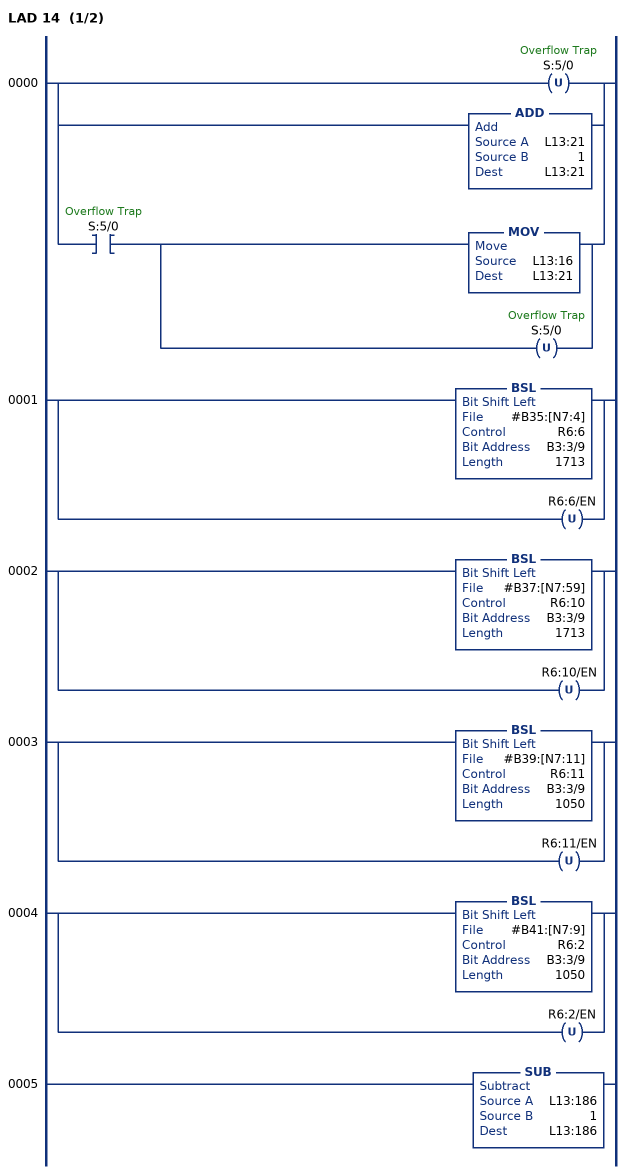
% Rung: 0 %
SOR BST OTU S:5/0 NXB ADD L13:21 1 L13:21 NXB XIC S:5/0 BST MOV L13:16 L13:21 NXB OTU S:5/0 BND BND EOR
%   S:5/0  "Overflow Trap" %
% Rung: 1 %
SOR BST BSL #B35:[N7:4] R6:6 B3:3/9 1713 NXB OTU R6:6/EN BND EOR
% Rung: 2 %
SOR BST BSL #B37:[N7:59] R6:10 B3:3/9 1713 NXB OTU R6:10/EN BND EOR
% Rung: 3 %
SOR BST BSL #B39:[N7:11] R6:11 B3:3/9 1050 NXB OTU R6:11/EN BND EOR
% Rung: 4 %
SOR BST BSL #B41:[N7:9] R6:2 B3:3/9 1050 NXB OTU R6:2/EN BND EOR
% Rung: 5 %
SOR SUB L13:186 1 L13:186 EOR

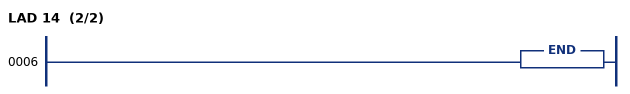
% Rung: 6 %
SOR END EOR

LADDER 81
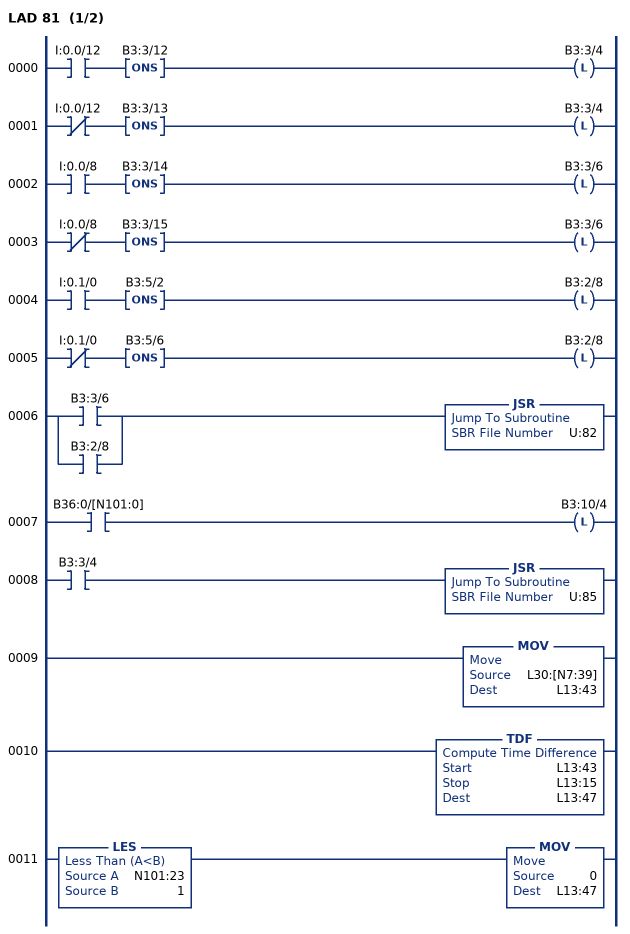
% Rung: 0 %
SOR XIC I:0.0/12 ONS B3:3/12 OTL B3:3/4 EOR
% Rung: 1 %
SOR XIO I:0.0/12 ONS B3:3/13 OTL B3:3/4 EOR
% Rung: 2 %
SOR XIC I:0.0/8 ONS B3:3/14 OTL B3:3/6 EOR
% Rung: 3 %
SOR XIO I:0.0/8 ONS B3:3/15 OTL B3:3/6 EOR
% Rung: 4 %
SOR XIC I:0.1/0 ONS B3:5/2 OTL B3:2/8 EOR
% Rung: 5 %
SOR XIO I:0.1/0 ONS B3:5/6 OTL B3:2/8 EOR
% Rung: 6 %
SOR BST XIC B3:3/6 NXB XIC B3:2/8 BND JSR U:82 EOR
% Rung: 7 %
SOR XIC B36:0/[N101:0] OTL B3:10/4 EOR
% Rung: 8 %
SOR XIC B3:3/4 JSR U:85 EOR
% Rung: 9 %
SOR MOV L30:[N7:39] L13:43 EOR
% Rung: 10 %
SOR TDF L13:43 L13:15 L13:47 EOR
% Rung: 11 %
SOR LES N101:23 1 MOV 0 L13:47 EOR

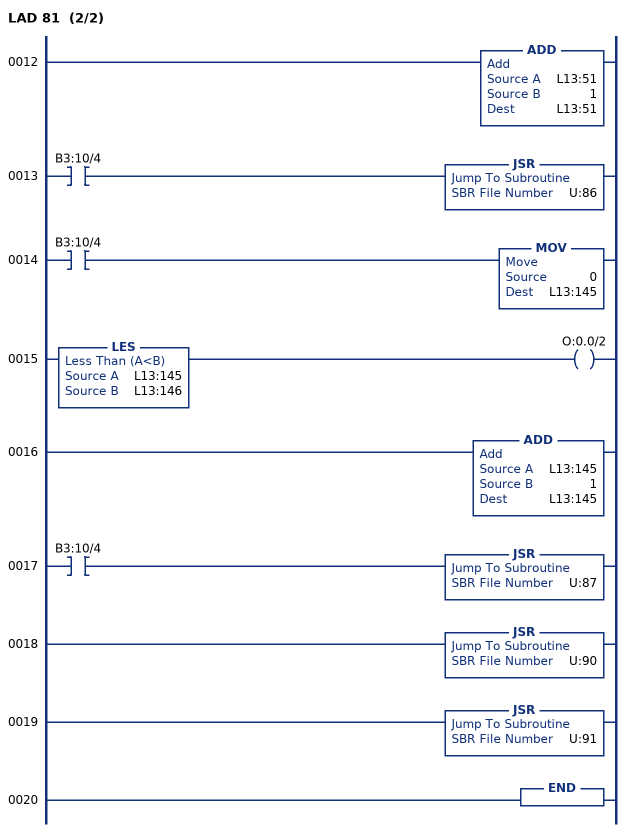
% Rung: 12 %
SOR ADD L13:51 1 L13:51 EOR
% Rung: 13 %
SOR XIC B3:10/4 JSR U:86 EOR
% Rung: 14 %
SOR XIC B3:10/4 MOV 0 L13:145 EOR
% Rung: 15 %
SOR LES L13:145 L13:146 OTE O:0.0/2 EOR
% Rung: 16 %
SOR ADD L13:145 1 L13:145 EOR
% Rung: 17 %
SOR XIC B3:10/4 JSR U:87 EOR
% Rung: 18 %
SOR JSR U:90 EOR
% Rung: 19 %
SOR JSR U:91 EOR
% Rung: 20 %
SOR END EOR

LADDER 82
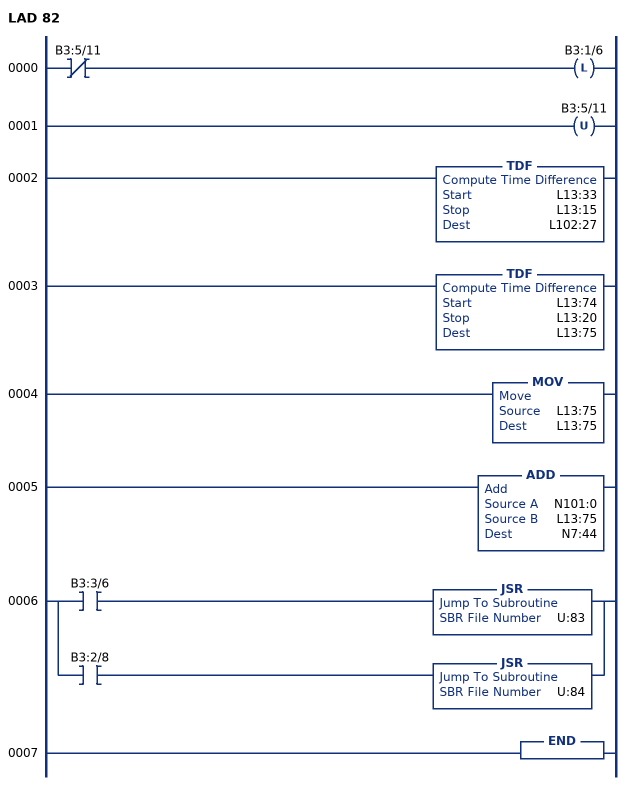
% Rung: 0 %
SOR XIO B3:5/11 OTL B3:1/6 EOR
% Rung: 1 %
SOR OTU B3:5/11 EOR
% Rung: 2 %
SOR TDF L13:33 L13:15 L102:27 EOR
% Rung: 3 %
SOR TDF L13:74 L13:20 L13:75 EOR
% Rung: 4 %
SOR MOV L13:75 L13:75 EOR
% Rung: 5 %
SOR ADD N101:0 L13:75 N7:44 EOR
% Rung: 6 %
SOR BST XIC B3:3/6 JSR U:83 NXB XIC B3:2/8 JSR U:84 BND EOR
% Rung: 7 %
SOR END EOR

LADDER 83
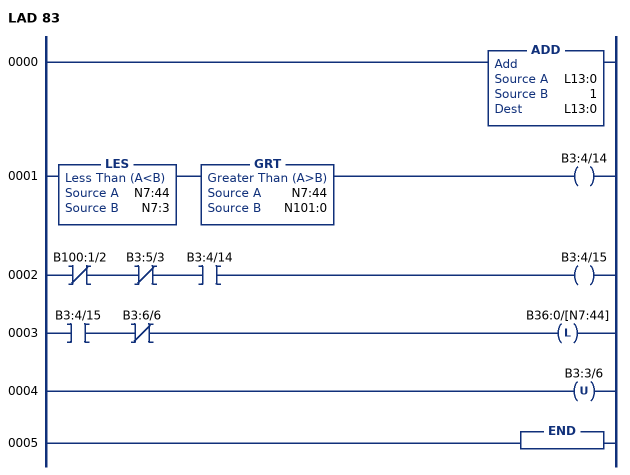
% Rung: 0 %
SOR ADD L13:0 1 L13:0 EOR
% Rung: 1 %
SOR LES N7:44 N7:3 GRT N7:44 N101:0 OTE B3:4/14 EOR
% Rung: 2 %
SOR XIO B100:1/2 XIO B3:5/3 XIC B3:4/14 OTE B3:4/15 EOR
% Rung: 3 %
SOR XIC B3:4/15 XIO B3:6/6 OTL B36:0/[N7:44] EOR
% Rung: 4 %
SOR OTU B3:3/6 EOR
% Rung: 5 %
SOR END EOR

LADDER 84
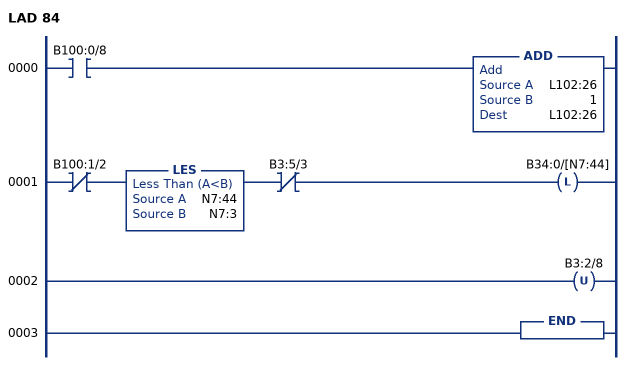
% Rung: 0 %
SOR XIC B100:0/8 ADD L102:26 1 L102:26 EOR
% Rung: 1 %
SOR XIO B100:1/2 LES N7:44 N7:3 XIO B3:5/3 OTL B34:0/[N7:44] EOR
% Rung: 2 %
SOR OTU B3:2/8 EOR
% Rung: 3 %
SOR END EOR

LADDER 85
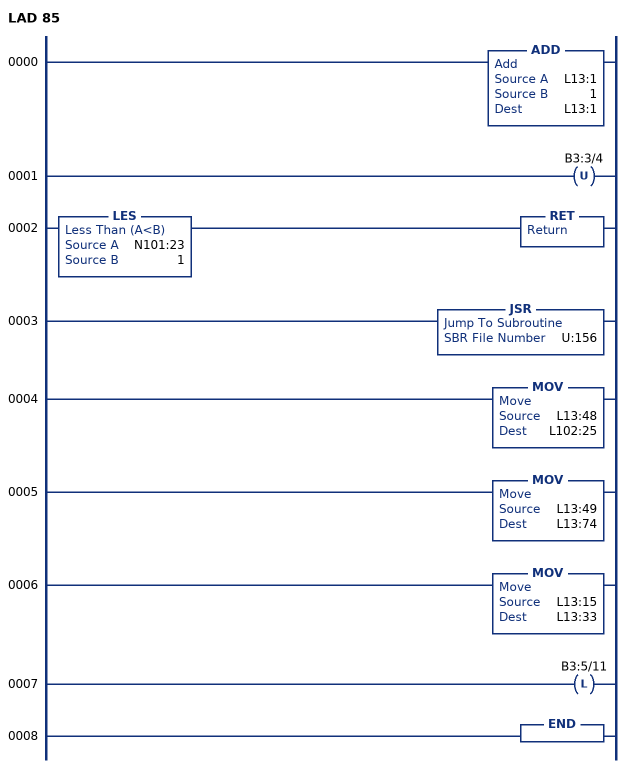
% Rung: 0 %
SOR ADD L13:1 1 L13:1 EOR
% Rung: 1 %
SOR OTU B3:3/4 EOR
% Rung: 2 %
SOR LES N101:23 1 RET EOR
% Rung: 3 %
SOR JSR U:156 EOR
% Rung: 4 %
SOR MOV L13:48 L102:25 EOR
% Rung: 5 %
SOR MOV L13:49 L13:74 EOR
% Rung: 6 %
SOR MOV L13:15 L13:33 EOR
% Rung: 7 %
SOR OTL B3:5/11 EOR
% Rung: 8 %
SOR END EOR

LADDER 86
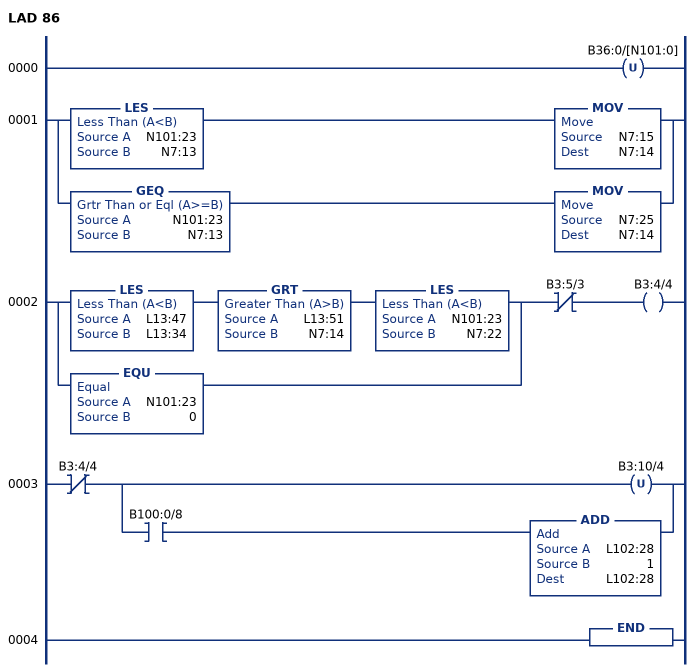
% Rung: 0 %
SOR OTU B36:0/[N101:0] EOR
% Rung: 1 %
SOR BST LES N101:23 N7:13 MOV N7:15 N7:14 NXB GEQ N101:23 N7:13 MOV N7:25 N7:14 BND EOR
% Rung: 2 %
SOR BST LES L13:47 L13:34 GRT L13:51 N7:14 LES N101:23 N7:22 NXB EQU N101:23 0 BND XIO B3:5/3 OTE B3:4/4 EOR
% Rung: 3 %
SOR XIO B3:4/4 BST OTU B3:10/4 NXB XIC B100:0/8 ADD L102:28 1 L102:28 BND EOR
% Rung: 4 %
SOR END EOR

LADDER 87
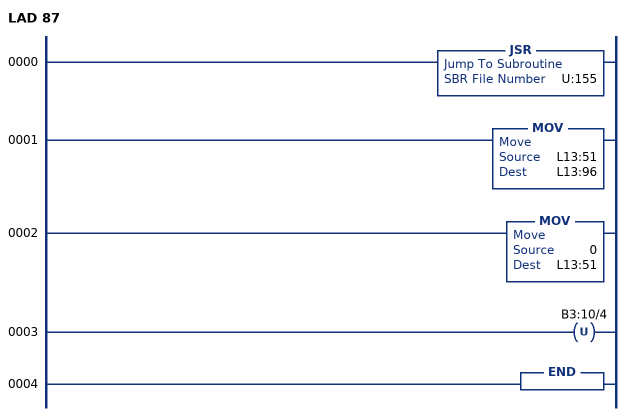
% Rung: 0 %
SOR JSR U:155 EOR
% Rung: 1 %
SOR MOV L13:51 L13:96 EOR
% Rung: 2 %
SOR MOV 0 L13:51 EOR
% Rung: 3 %
SOR OTU B3:10/4 EOR
% Rung: 4 %
SOR END EOR

LADDER 90
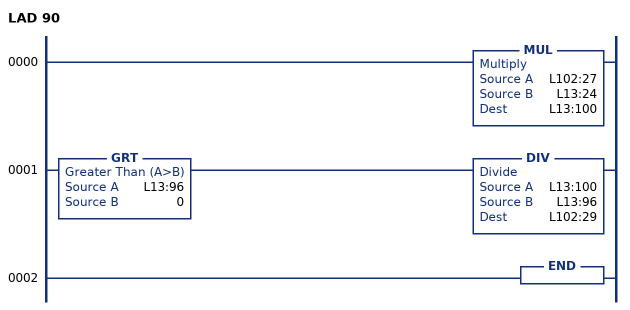
% Rung: 0 %
SOR MUL L102:27 L13:24 L13:100 EOR
% Rung: 1 %
SOR GRT L13:96 0 DIV L13:100 L13:96 L102:29 EOR
% Rung: 2 %
SOR END EOR

LADDER 91
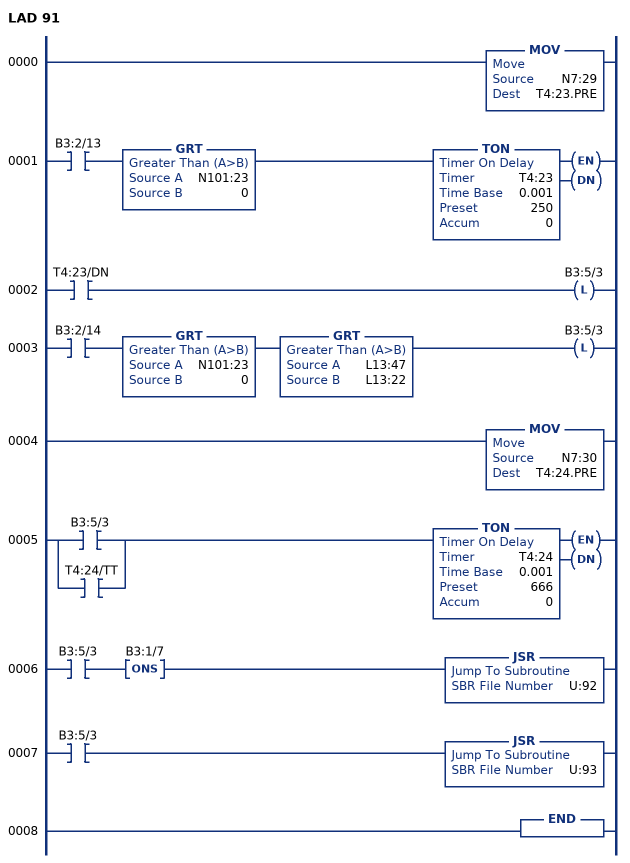
% Rung: 0 %
SOR MOV N7:29 T4:23.PRE EOR
% Rung: 1 %
SOR XIC B3:2/13 GRT N101:23 0 TON T4:23 0.001 250 0 EOR
% Rung: 2 %
SOR XIC T4:23/DN OTL B3:5/3 EOR
% Rung: 3 %
SOR XIC B3:2/14 GRT N101:23 0 GRT L13:47 L13:22 OTL B3:5/3 EOR
% Rung: 4 %
SOR MOV N7:30 T4:24.PRE EOR
% Rung: 5 %
SOR BST XIC B3:5/3 NXB XIC T4:24/TT BND TON T4:24 0.001 666 0 EOR
% Rung: 6 %
SOR XIC B3:5/3 ONS B3:1/7 JSR U:92 EOR
% Rung: 7 %
SOR XIC B3:5/3 JSR U:93 EOR
% Rung: 8 %
SOR END EOR

LADDER 92
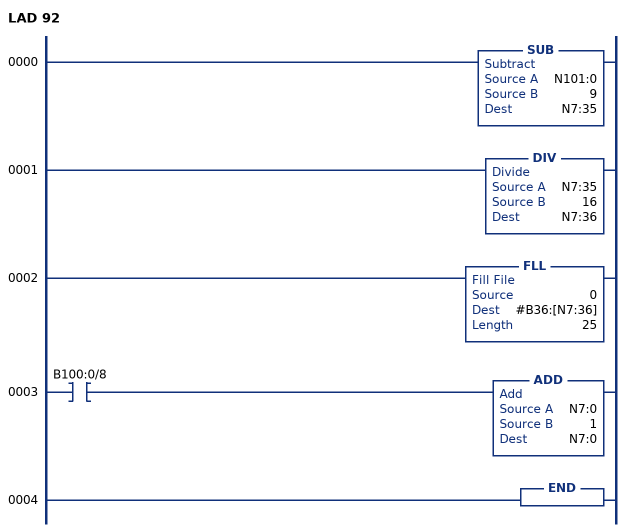
% Rung: 0 %
SOR SUB N101:0 9 N7:35 EOR
% Rung: 1 %
SOR DIV N7:35 16 N7:36 EOR
% Rung: 2 %
SOR FLL 0 #B36:[N7:36] 25 EOR
% Rung: 3 %
SOR XIC B100:0/8 ADD N7:0 1 N7:0 EOR
% Rung: 4 %
SOR END EOR

LADDER 93
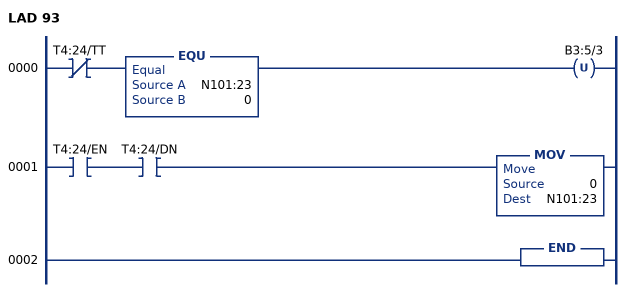
% Rung: 0 %
SOR XIO T4:24/TT EQU N101:23 0 OTU B3:5/3 EOR
% Rung: 1 %
SOR XIC T4:24/EN XIC T4:24/DN MOV 0 N101:23 EOR
% Rung: 2 %
SOR END EOR

LADDER 94
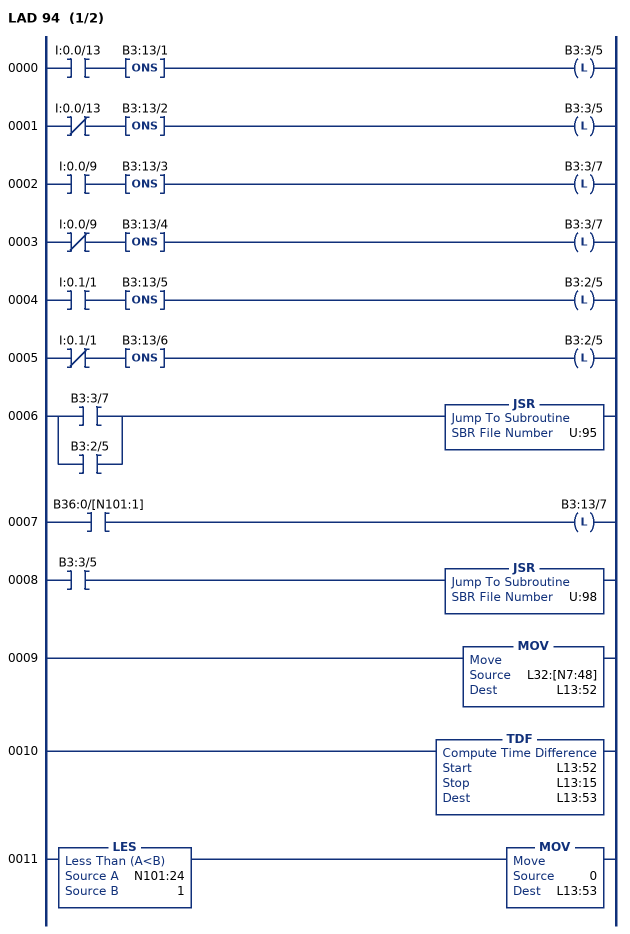
% Rung: 0 %
SOR XIC I:0.0/13 ONS B3:13/1 OTL B3:3/5 EOR
% Rung: 1 %
SOR XIO I:0.0/13 ONS B3:13/2 OTL B3:3/5 EOR
% Rung: 2 %
SOR XIC I:0.0/9 ONS B3:13/3 OTL B3:3/7 EOR
% Rung: 3 %
SOR XIO I:0.0/9 ONS B3:13/4 OTL B3:3/7 EOR
% Rung: 4 %
SOR XIC I:0.1/1 ONS B3:13/5 OTL B3:2/5 EOR
% Rung: 5 %
SOR XIO I:0.1/1 ONS B3:13/6 OTL B3:2/5 EOR
% Rung: 6 %
SOR BST XIC B3:3/7 NXB XIC B3:2/5 BND JSR U:95 EOR
% Rung: 7 %
SOR XIC B36:0/[N101:1] OTL B3:13/7 EOR
% Rung: 8 %
SOR XIC B3:3/5 JSR U:98 EOR
% Rung: 9 %
SOR MOV L32:[N7:48] L13:52 EOR
% Rung: 10 %
SOR TDF L13:52 L13:15 L13:53 EOR
% Rung: 11 %
SOR LES N101:24 1 MOV 0 L13:53 EOR

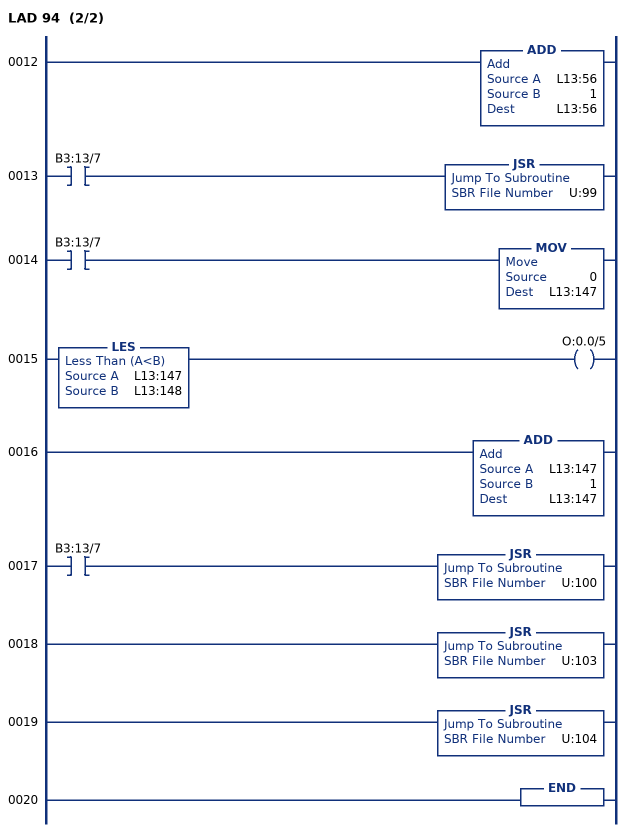
% Rung: 12 %
SOR ADD L13:56 1 L13:56 EOR
% Rung: 13 %
SOR XIC B3:13/7 JSR U:99 EOR
% Rung: 14 %
SOR XIC B3:13/7 MOV 0 L13:147 EOR
% Rung: 15 %
SOR LES L13:147 L13:148 OTE O:0.0/5 EOR
% Rung: 16 %
SOR ADD L13:147 1 L13:147 EOR
% Rung: 17 %
SOR XIC B3:13/7 JSR U:100 EOR
% Rung: 18 %
SOR JSR U:103 EOR
% Rung: 19 %
SOR JSR U:104 EOR
% Rung: 20 %
SOR END EOR

LADDER 95
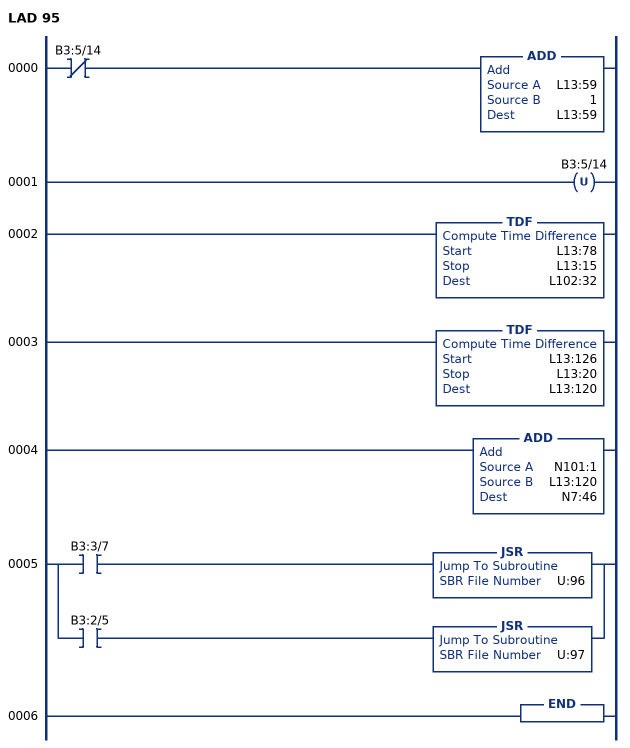
% Rung: 0 %
SOR XIO B3:5/14 ADD L13:59 1 L13:59 EOR
% Rung: 1 %
SOR OTU B3:5/14 EOR
% Rung: 2 %
SOR TDF L13:78 L13:15 L102:32 EOR
% Rung: 3 %
SOR TDF L13:126 L13:20 L13:120 EOR
% Rung: 4 %
SOR ADD N101:1 L13:120 N7:46 EOR
% Rung: 5 %
SOR BST XIC B3:3/7 JSR U:96 NXB XIC B3:2/5 JSR U:97 BND EOR
% Rung: 6 %
SOR END EOR

LADDER 96
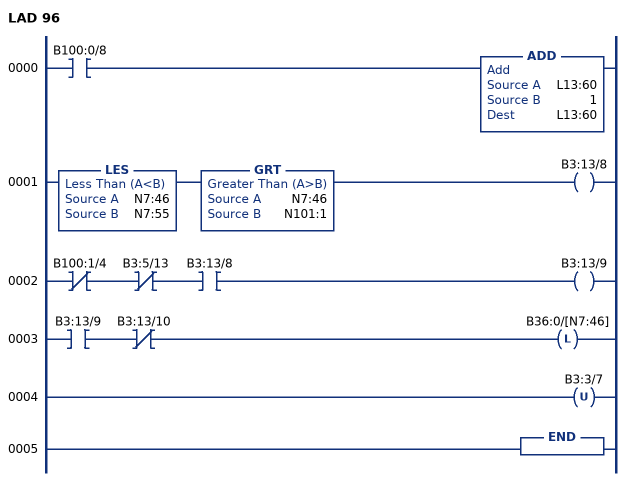
% Rung: 0 %
SOR XIC B100:0/8 ADD L13:60 1 L13:60 EOR
% Rung: 1 %
SOR LES N7:46 N7:55 GRT N7:46 N101:1 OTE B3:13/8 EOR
% Rung: 2 %
SOR XIO B100:1/4 XIO B3:5/13 XIC B3:13/8 OTE B3:13/9 EOR
% Rung: 3 %
SOR XIC B3:13/9 XIO B3:13/10 OTL B36:0/[N7:46] EOR
% Rung: 4 %
SOR OTU B3:3/7 EOR
% Rung: 5 %
SOR END EOR

LADDER 97
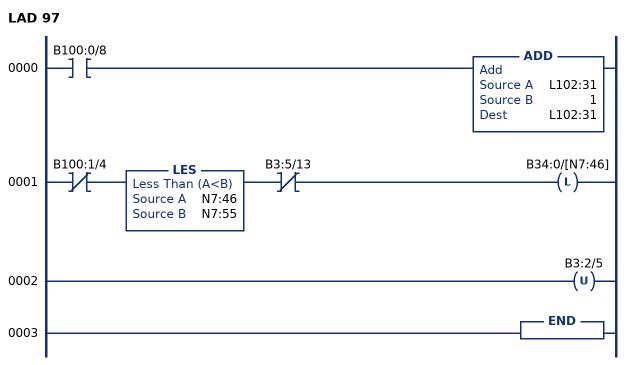
% Rung: 0 %
SOR XIC B100:0/8 ADD L102:31 1 L102:31 EOR
% Rung: 1 %
SOR XIO B100:1/4 LES N7:46 N7:55 XIO B3:5/13 OTL B34:0/[N7:46] EOR
% Rung: 2 %
SOR OTU B3:2/5 EOR
% Rung: 3 %
SOR END EOR

LADDER 98
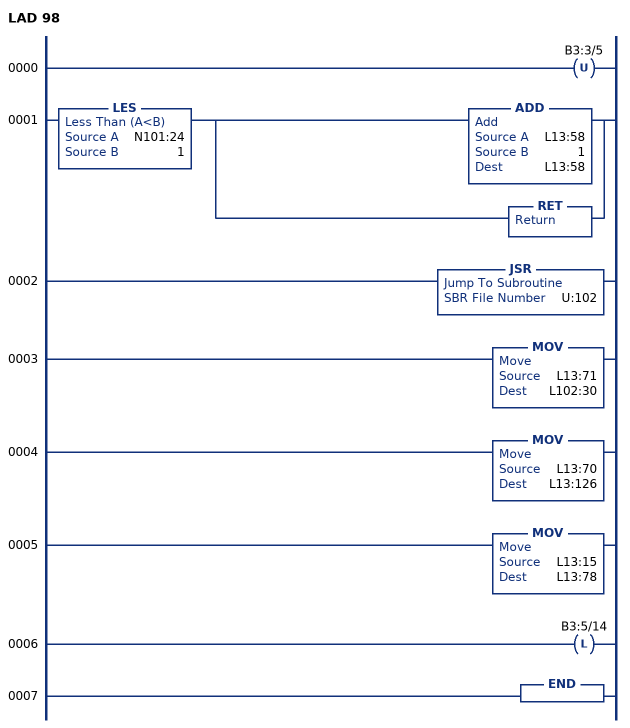
% Rung: 0 %
SOR OTU B3:3/5 EOR
% Rung: 1 %
SOR LES N101:24 1 BST ADD L13:58 1 L13:58 NXB RET BND EOR
% Rung: 2 %
SOR JSR U:102 EOR
% Rung: 3 %
SOR MOV L13:71 L102:30 EOR
% Rung: 4 %
SOR MOV L13:70 L13:126 EOR
% Rung: 5 %
SOR MOV L13:15 L13:78 EOR
% Rung: 6 %
SOR OTL B3:5/14 EOR
% Rung: 7 %
SOR END EOR

LADDER 99
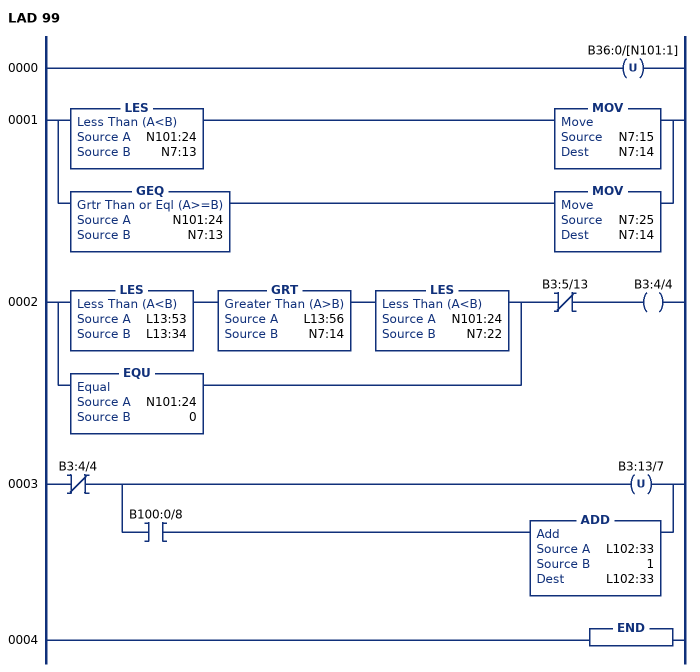
% Rung: 0 %
SOR OTU B36:0/[N101:1] EOR
% Rung: 1 %
SOR BST LES N101:24 N7:13 MOV N7:15 N7:14 NXB GEQ N101:24 N7:13 MOV N7:25 N7:14 BND EOR
% Rung: 2 %
SOR BST LES L13:53 L13:34 GRT L13:56 N7:14 LES N101:24 N7:22 NXB EQU N101:24 0 BND XIO B3:5/13 OTE B3:4/4 EOR
% Rung: 3 %
SOR XIO B3:4/4 BST OTU B3:13/7 NXB XIC B100:0/8 ADD L102:33 1 L102:33 BND EOR
% Rung: 4 %
SOR END EOR

LADDER 100
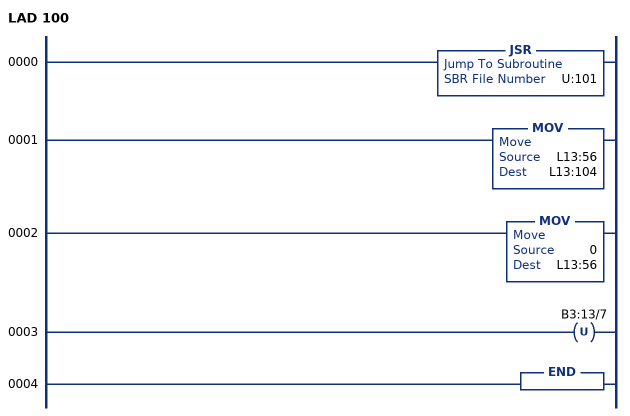
% Rung: 0 %
SOR JSR U:101 EOR
% Rung: 1 %
SOR MOV L13:56 L13:104 EOR
% Rung: 2 %
SOR MOV 0 L13:56 EOR
% Rung: 3 %
SOR OTU B3:13/7 EOR
% Rung: 4 %
SOR END EOR

LADDER 101
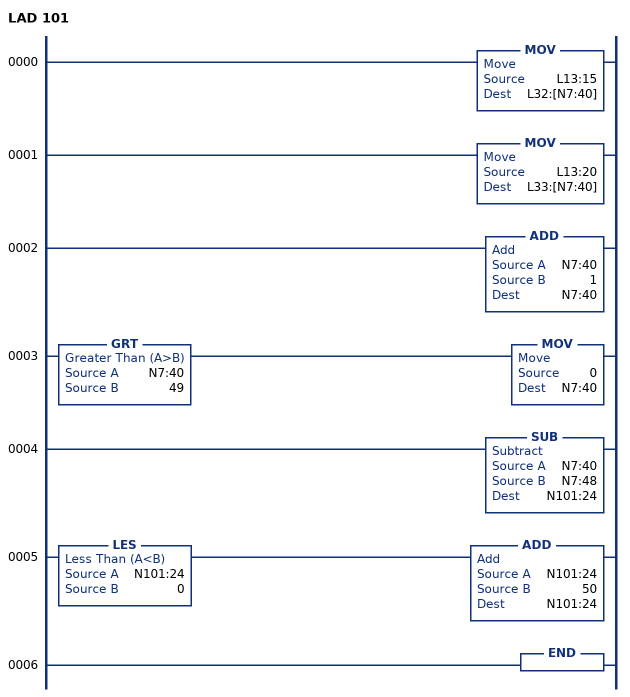
% Rung: 0 %
SOR MOV L13:15 L32:[N7:40] EOR
% Rung: 1 %
SOR MOV L13:20 L33:[N7:40] EOR
% Rung: 2 %
SOR ADD N7:40 1 N7:40 EOR
% Rung: 3 %
SOR GRT N7:40 49 MOV 0 N7:40 EOR
% Rung: 4 %
SOR SUB N7:40 N7:48 N101:24 EOR
% Rung: 5 %
SOR LES N101:24 0 ADD N101:24 50 N101:24 EOR
% Rung: 6 %
SOR END EOR

LADDER 102
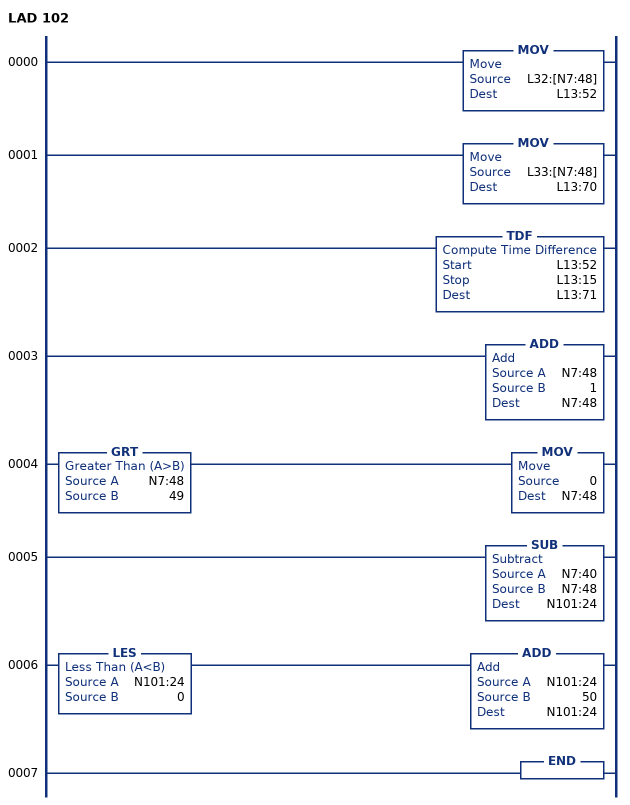
% Rung: 0 %
SOR MOV L32:[N7:48] L13:52 EOR
% Rung: 1 %
SOR MOV L33:[N7:48] L13:70 EOR
% Rung: 2 %
SOR TDF L13:52 L13:15 L13:71 EOR
% Rung: 3 %
SOR ADD N7:48 1 N7:48 EOR
% Rung: 4 %
SOR GRT N7:48 49 MOV 0 N7:48 EOR
% Rung: 5 %
SOR SUB N7:40 N7:48 N101:24 EOR
% Rung: 6 %
SOR LES N101:24 0 ADD N101:24 50 N101:24 EOR
% Rung: 7 %
SOR END EOR

LADDER 103
